{attribute 'GeneratedUsingTerminal: EL2522-0000-0017'}
{attribute addProperty BoxType "EL2522-0000-0017"}
{attribute addProperty Id "StatusAT %I*Status_B83811715"}
{attribute addProperty CRC "3773501672"}
{attribute addProperty Size "5"}
TYPE PTO_Status_Channel_E0EB10E8 :
STRUCT
	{attribute addProperty Name "Status"}
	Status AT %I* : Status_B8381171;
END_STRUCT
END_TYPE

(* stored: Version 1.2.0.0, ProductVersion 3.1.4024.9
   DUT PTO_Status_Channel_E0EB10E8: Id {e0ce9a02-2aac-40a0-8a9a-39e01bdb988a} *)
